Staubli VAL3: onF8Event.pgx

program onF8Event()
  local string l_sMessage
begin
  // look if the bButton is enable
  if bButton[7]
    //
  endIf
end
